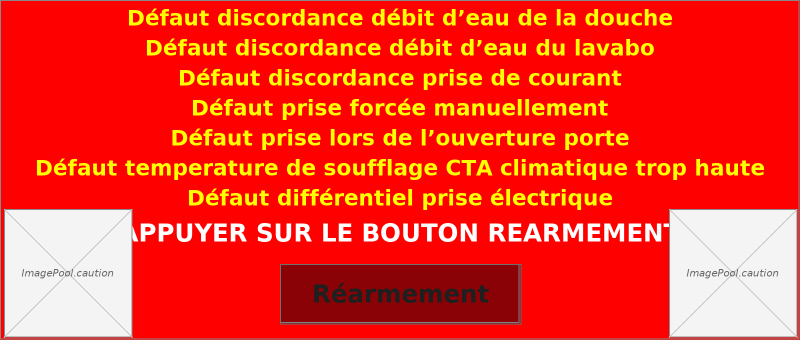
VISUALIZATION PopUp_Alarms  // 800x340
    RoundedRectangle (0,3 800x30), "Défaut discordance débit d’eau de la douche", invisible if: NOT Defaut_Discord_Deb_Eau_Douche
    Button (280,264 241x60), "Réarmement", invisible if: NOT Condi_Affich_Rearm
        OnMouseDown: toggle Cmd_Rearmement
    RoundedRectangle (0,208 800x50), "APPUYER SUR LE BOUTON REARMEMENT"
    Image (4,209 128x128), image: ImagePool.caution
    Image (669,209 128x128), image: ImagePool.caution
    RoundedRectangle (0,33 800x30), "Défaut discordance débit d’eau du lavabo", invisible if: NOT Defaut_Discord_Deb_Eau_Lavabo
    RoundedRectangle (0,63 800x30), "Défaut discordance prise de courant", invisible if: NOT Defaut_Discord_PC_Cab
    RoundedRectangle (0,93 800x30), "Défaut prise forcée manuellement", invisible if: NOT Def_Discord_Alim_Prise
    RoundedRectangle (0,123 800x30), "Défaut prise lors de l’ouverture porte", invisible if: NOT Def_Prise_Porte_Ouverte
    RoundedRectangle (0,183 800x30), "Défaut différentiel prise électrique", invisible if: NOT Defaut_Differentiel_Prise_Elec
    RoundedRectangle (0,153 800x30), "Défaut temperature de soufflage CTA climatique trop haute", invisible if: NOT Defaut_Thermostat_Secu
END_VISUALIZATION

(* stored: Version 1.1.0.1, ProductVersion 3.1.4024.15
   Visu PopUp_Alarms: Id {dd629bc1-d7c0-4aef-a19e-22c642a82325} *)
